{attribute 'qualified_only'}
{attribute 'strict'}
TYPE FanTypes :
(
	EBM := 0, Gebhardt
);
END_TYPE

(* stored: Version 1.1.0.1, ProductVersion 3.1.4024.6
   DUT FanTypes: Id {358019fd-dbbb-4482-a66b-d2c026f38d79} *)
